// TIA Portal V16 export
// export: Created 2024-12-03T15:41:46.1891708Z, ExportSetting WithReadOnly, DisplayName Totally Integrated Automation Portal, DisplayVersion V16 Update 6, DisplayName TIA Portal Version Control Interface, DisplayVersion V16 Update 2, DisplayName TIA Portal Openness, DisplayVersion V16 Update 6, DisplayName TIA Portal Teamcenter Gateway, DisplayVersion V16, DisplayName SINAMICS Startdrive Advanced, DisplayVersion V16 Update 5, DisplayName SINAMICS Startdrive G130, G150, S120, S150, SINAMICS MV, S210, DisplayVersion V16 Update 5, DisplayName SINAMICS Startdrive G110M, G120, G120C, G120D, G120P, G115D, DisplayVersion V16 Update 5, DisplayName STEP 7 Professional, DisplayVersion V16 Update 6, DisplayName STEP 7 Safety, DisplayVersion V16, DisplayName WinCC Advanced / Unified PC, DisplayVersion V16 Update 6
TYPE "appButtons_UDT"
// stored: CreationDate 2021-07-13T07:41:36.2278727Z, InterfaceModifiedDate 2021-03-12T11:44:15.2886107Z, IsConsistent true, LibraryConformanceStatus The object is library-conformant., ModifiedDate 2021-07-03T12:49:45.6036717Z
   STRUCT
      reset { S7_SetPoint := 'True'} : "HMIButton_UDT";
      StartAutoMode { S7_SetPoint := 'True'} : "HMIButton_UDT";
      ActivateManualMode { S7_SetPoint := 'True'} : "HMIButton_UDT";
      StopAutoMode { S7_SetPoint := 'True'} : "HMIButton_UDT";
      DeactivateManualMode { S7_SetPoint := 'True'} : "HMIButton_UDT";
      StartEmptyMode { S7_SetPoint := 'True'} : "HMIButton_UDT";
      StopEmptyMode { S7_SetPoint := 'True'} : "HMIButton_UDT";
      ActivateStandby { S7_SetPoint := 'True'} : "HMIButton_UDT";
   END_STRUCT;
END_TYPE
